FUNCTION_BLOCK FB_StepperMotor
VAR_INPUT
	nRail 	   : SINT := 0;
END_VAR
VAR
	pAxis : POINTER TO AXIS_REF;
	fRead : MC_ReadActualPosition;
    fbPower    : MC_Power;
    fbstop     : MC_Halt;
    fbMoveAbs  : MC_MoveAbsolute;
    fbhome     : MC_Home;
    fbRead     : MC_ReadActualPosition;               
    nErrID     : UDINT;               
    fbReset    : MC_Reset;
	eState	   : ENUM_StepperMotorState := LAS_Stepper_Uninitialized;    
END_VAR

METHOD CheckHardware : BOOL
VAR_INPUT
END_VAR
END_METHOD

METHOD FB_Init: BOOL
VAR_INPUT
    bInitRetains: BOOL; 
    bInCopyCode: BOOL;  
	init_axis : POINTER TO AXIS_REF;
END_VAR
pAxis := init_axis;
END_METHOD

METHOD GetPosition : BOOL
VAR
	pAlarmCondition : POINTER TO BOOL;
END_VAR
VAR_OUTPUT
	fCurrentPosition : LREAL;
END_VAR
Init(Axis := pAxis);
fRead(Axis := pAxis^, Enable := TRUE, Position => fCurrentPosition);

IF fRead.Busy THEN
	IF fRead.Error THEN
		pAlarmCondition := F_GetStepperAlarmCondition(nRail, 'UnableToReadPosition');
		IF pAlarmCondition <> 0 THEN
			pAlarmCondition^ := TRUE;
		END_IF
	END_IF

ELSE
	IF NOT fRead.Valid THEN
		fCurrentPosition := -1;
	END_IF
END_IF
END_METHOD

METHOD Home : INT
VAR_INPUT
    bExecute : BOOL;     
END_VAR
VAR
    Currentpos : LREAL;
	Currentpass : STRING := 'Fast';
    FastPass : ST_HomingOptions := (SearchVelocity := 50.0, SyncVelocity := 15.0);
    SlowPass : ST_HomingOptions := (SearchVelocity := 5.0, SyncVelocity := 2.0);
	ReferencePos : LREAL := 10.0;    
	bPreviousSwitchState: BOOL := FALSE;
	bFirstEdgeDetected: BOOL := FALSE;
	pAlarmCondition : POINTER TO BOOL;
END_VAR
Init(Axis := pAxis); //Keep actuator up
GetPosition(fCurrentPosition => Currentpos);

CASE eState OF
    LAS_Stepper_Idle:
        IF Currentpass = 'Fast' THEN
            fbHome(Axis := pAxis^, Execute := TRUE, HomingMode := 0, Position := ReferencePos, bCalibrationCam := NOT bSimulatedLimitSwitch, Options := FastPass);
            eState := LAS_Stepper_FastPass;
            
        ELSIF Currentpass = 'Slow' THEN
            fbHome(Axis := pAxis^, Execute := TRUE, HomingMode := 0, Position := ReferencePos, bCalibrationCam := NOT bSimulatedLimitSwitch, Options := SlowPass);
            eState := LAS_Stepper_SlowPass;
        END_IF
        
    LAS_Stepper_FastPass:
        fbHome(Axis := pAxis^, bCalibrationCam := NOT bSimulatedLimitSwitch);
        
        IF fbHome.Error THEN
			(*IF fbHome.ErrorID = 16#00004B0A THEN
				
				pAlarmCondition := F_GetStepperAlarmCondition(nRail, 'Homing_Interrupted');
				IF pAlarmCondition <> 0 THEN
					pAlarmCondition^ := TRUE;
				END_IF
				
				Home := -1;
				RETURN;
			END_IF*)
			
            eState := LAS_Stepper_Error;
            
			pAlarmCondition := F_GetStepperAlarmCondition(nRail, 'Homing_Failed');
			IF pAlarmCondition <> 0 THEN
				pAlarmCondition^ := TRUE;
			END_IF
				
            nErrID := fbHome.ErrorID;
            Home := -1;

        ELSIF fbHome.Done THEN
            fbHome(Axis := pAxis^, Execute := FALSE);
            eState := LAS_Stepper_WaitingForTrigger;
        END_IF
    
    LAS_Stepper_WaitingForTrigger: // Wait for the limit switch

        IF NOT bSimulatedLimitSwitch THEN

            fbHome(Axis := pAxis^, Execute := TRUE, HomingMode := 0, Position := ReferencePos, bCalibrationCam := NOT bSimulatedLimitSwitch, Options := SlowPass);
            eState := LAS_Stepper_SlowPass;
        END_IF
    
    LAS_Stepper_SlowPass:
        fbHome(Axis := pAxis^, bCalibrationCam := NOT bSimulatedLimitSwitch);
        
        IF fbHome.Error THEN
			(*IF fbHome.ErrorID = 16#00004B0A THEN
				
				pAlarmCondition := F_GetStepperAlarmCondition(nRail, 'Homing_Interrupted');
				IF pAlarmCondition <> 0 THEN
					pAlarmCondition^ := TRUE;
				END_IF
				
				Home := -1;
				RETURN;
			END_IF*)
			
            eState := LAS_Stepper_Error;
            
			pAlarmCondition := F_GetStepperAlarmCondition(nRail, 'Homing_Failed');
			IF pAlarmCondition <> 0 THEN
				pAlarmCondition^ := TRUE;
			END_IF
			
            nErrID := fbHome.ErrorID;
            Home := -1;
			
        ELSIF fbHome.Done THEN
            fbHome(Axis := pAxis^, Execute := FALSE);
            Currentpass := 'Fast';
            Home := 1; 
            eState := LAS_Stepper_Idle;
        END_IF
    
    LAS_Stepper_Error:
        Home := -1;
        
END_CASE
END_METHOD

METHOD Init : BOOL
VAR_INPUT
	Axis : POINTER TO AXIS_REF;  
END_VAR

VAR
	pAlarmCondition : POINTER TO BOOL;
END_VAR
pAxis := Axis; 

CASE eState OF 
    LAS_Stepper_Uninitialized:
        fbPower(Axis := pAxis^, Enable := TRUE, Enable_positive := TRUE, Enable_Negative := TRUE);
        
		IF fbPower.Status THEN
			Init := TRUE; 
			eState := LAS_Stepper_Idle;
			nErrID := 0;
			//Enable := FALSE;
			
		ELSIF fbPower.Error THEN	
			nErrID := fbPower.ErrorID;
			eState := LAS_Stepper_Error;
			
			pAlarmCondition := F_GetStepperAlarmCondition(nRail, 'PowerUp_Failed');
			IF pAlarmCondition <> 0 THEN
				pAlarmCondition^ := TRUE;
			END_IF
			
			Init := FALSE;
			//Enable := FALSE;
		END_IF
      
	  ELSE
	  	
	  	fbPower(Axis := pAxis^, Enable := TRUE, Enable_positive := TRUE, Enable_Negative := TRUE);
		IF fbPower.Error THEN	
			nErrID := fbPower.ErrorID;
			eState := LAS_Stepper_Error;
			
			pAlarmCondition := F_GetStepperAlarmCondition(nRail, 'PowerUp_Failed');
			IF pAlarmCondition <> 0 THEN
				pAlarmCondition^ := TRUE;
			END_IF
			
			Init := FALSE;
			//Enable := FALSE;
		END_IF
				
END_CASE
END_METHOD

METHOD MoveToPosition : INT
VAR_INPUT
    fPosition : LREAL;  // Target position
    fVelocity : LREAL := 100.0;  // Velocity in mm/s
    fAccel    : LREAL := 500.0;  // Acceleration in mm/s²
    fDecel    : LREAL := 500.0;  // Deceleration in mm/s²
END_VAR

VAR
	pAlarmCondition : POINTER TO BOOL;
END_VAR
MoveToPosition := 0;
Init(Axis := pAxis);

CASE eState OF
	LAS_Stepper_Idle:
		fbMoveAbs(Axis := pAxis^, Execute := TRUE, Position := fPosition, 
          Velocity := fVelocity, Acceleration := fAccel, Deceleration := fDecel);
	
		eState := LAS_Stepper_Moving;
		
	LAS_Stepper_Moving:
		IF fbMoveAbs.Busy THEN
			fbMoveAbs(Axis := pAxis^);
			IF fbMoveAbs.Error THEN
				eState := LAS_Stepper_Error;
				
				nErrID := fbMoveAbs.ErrorID;
				
				pAlarmCondition := F_GetStepperAlarmCondition(nRail, 'Motion_Failed');
				IF pAlarmCondition <> 0 THEN
					pAlarmCondition^ := TRUE;
				END_IF
				
				MoveToPosition := -1;
			END_IF
		
		ELSIF fbMoveAbs.CommandAborted THEN
			eState := LAS_Stepper_Error;
			
			pAlarmCondition := F_GetStepperAlarmCondition(nRail, 'Motion_Interrupted');
			IF pAlarmCondition <> 0 THEN
				pAlarmCondition^ := TRUE;
			END_IF
				
			fbMoveAbs(Axis := pAxis^, Execute := FALSE);
			MoveToPosition := -1;
			
		ELSIF fbMoveAbs.Done THEN
			eState := LAS_Stepper_Idle;
			fbMoveAbs(Axis := pAxis^, Execute := FALSE);
			MoveToPosition := 1; 
			nErrID := 0;
		END_IF
	
	LAS_Stepper_Error:
		MoveToPosition := -1; 
		
END_CASE
END_METHOD

METHOD Reset : INT
VAR_INPUT
    bExecute : BOOL;
END_VAR

VAR
	i : UINT;
	pAlarmCondition : POINTER TO BOOL;
END_VAR
Reset := 0;
Init(Axis := pAxis);

IF eState = LAS_Stepper_Error THEN
	fbReset(Axis := pAxis^, Execute := bExecute);
	
	IF fbReset.Busy THEN 
		IF fbReset.Error THEN
			
		eState := LAS_Stepper_Error;
		nErrID := fbReset.ErrorID;
		
		pAlarmCondition := F_GetStepperAlarmCondition(nRail, 'Reset_Failed');
		IF pAlarmCondition <> 0 THEN
			pAlarmCondition^ := TRUE;
		END_IF
		
		Reset := -1;
		END_IF
	
	ELSIF fbReset.Done THEN
		Reset := 1;
		
		IF fbPower.Status THEN
			eState := LAS_Stepper_Idle;					
		ELSE
			eState := LAS_Stepper_Uninitialized;
		END_IF
		
	END_IF
END_IF
END_METHOD

METHOD Stop : INT
VAR_INPUT
    bEnable : BOOL;
	fDecel    : LREAL := 500.0;
END_VAR

VAR
	pAlarmCondition : POINTER TO BOOL;
END_VAR
Stop := 0;
Init(Axis := pAxis);

CASE eState OF
    LAS_Stepper_Idle:
        // Already stopped
        Stop := 1;
        
    LAS_Stepper_Moving:
        fbStop(Axis := pAxis^, Execute := bEnable, Deceleration := fDecel);
              
		IF fbStop.Error THEN
			fbStop(Axis := pAxis^, Execute := FALSE);
			eState := LAS_Stepper_Error;
			nErrID := fbStop.ErrorID;
			
			pAlarmCondition := F_GetStepperAlarmCondition(nRail, 'Stop_Failed');
			IF pAlarmCondition <> 0 THEN
				pAlarmCondition^ := TRUE;
			END_IF
			
			Stop := -1;
            
        ELSIF fbStop.Done THEN
			fbStop(Axis := pAxis^, Execute := FALSE);
			fbMoveAbs(Axis := pAxis^, Execute := FALSE);
            eState := LAS_Stepper_Idle;
            Stop := 1; 
            nErrID := 0;
		END_IF
    
    LAS_Stepper_FastPass, LAS_Stepper_SlowPass, LAS_Stepper_WaitingForTrigger :
	
	   fbStop(Axis := pAxis^, Execute := TRUE, Deceleration := fDecel);
	   
	   IF fbStop.Done THEN
		   fbStop(Axis := pAxis^, Execute := FALSE);
		   fbHome(Axis := pAxis^, Execute := FALSE);
		   fbReset(Axis := pAxis^, Execute := TRUE);
		   IF fbReset.Done THEN
		       fbReset(Axis := pAxis^, Execute := FALSE);
			   eState := LAS_Stepper_Idle;
		   	   Stop   := 1;          
	   	   END_IF
	   ELSIF fbStop.Error THEN
			eState := LAS_Stepper_Error;
			nErrID := fbStop.ErrorID;
			Stop   := -1;
	   END_IF
    
    LAS_Stepper_Error:
        Stop := -1;        
        
    ELSE
        // Unknown state
        fbStop(Axis := pAxis^, Execute := bEnable, Deceleration := fDecel);
        IF fbStop.Done THEN
            eState := LAS_Stepper_Idle;
            Stop := 1;
        ELSIF fbStop.Error THEN
            eState := LAS_Stepper_Error;
            nErrID := fbStop.ErrorID;
			
			pAlarmCondition := F_GetStepperAlarmCondition(nRail, 'Stop_Failed');
			IF pAlarmCondition <> 0 THEN
				pAlarmCondition^ := TRUE;
			END_IF
			
            Stop := -1;
        END_IF
        
END_CASE
END_METHOD

END_FUNCTION_BLOCK

(* stored: Version 1.1.0.1, ProductVersion 3.1.4026.11
   POU FB_StepperMotor: Id {bbe3d249-0f45-4d4f-9e26-26a436162bb5}, SpecialFunc None
   Method CheckHardware: Id {9483b802-41e4-45b6-80c4-0c5089e14c23}
   Method FB_Init: Id {aae538f2-84d5-46d9-a4e2-9cefceb9bd59}
   Method GetPosition: Id {c99d767f-ea4a-49f6-ba95-aa6815963f09}
   Method Home: Id {8276e0ce-98e0-421a-babf-511ef600c743}
   Method Init: Id {fa5103ef-9b92-4848-8e64-2a4a389deecc}
   Method MoveToPosition: Id {59187d53-eaea-489c-80e7-2ef214427a40}
   Method Reset: Id {185c3e3a-adea-4170-9d64-3a4611a9e6c3}
   Method Stop: Id {9b515f94-46a2-4ab1-aca0-af2dcdfe9f04} *)
